Staubli VAL3: default.pjx

--- default.pjx ---
Parameters version=s7.2.1 stackSize=5000 millimeterUnit=true
Data file=default.dtx
Library alias=io path=Disk://io/io.pjx

--- default.dtx ---
public num nDoneCycle
public num nDoneEnd
public num nDoneStart
public num nTime
public num nTotalCycle
public num nTotalEnd = 1
public num nTotalStart = 1
public num nType = 1
public string sLoadEnd
public string sLoadProg
public string sLoadStart
public bool bLoop = true
